// TIA Portal V17 export
// export: Created 2022-02-03T14:45:11.768442Z, ExportSetting WithDefaults, DisplayName Totally Integrated Automation Portal, DisplayVersion V17, DisplayName TIA Portal Openness, DisplayVersion V17, DisplayName TIA Portal Version Control Interface, DisplayVersion V17, DisplayName SINAMICS Startdrive Advanced, DisplayVersion V17, DisplayName SINAMICS Startdrive G130, G150, S120, S150, SINAMICS MV, S210, DisplayVersion V17, DisplayName SINAMICS Startdrive G110M, G120, G120C, G120D, G120P, G115D, DisplayVersion V17, DisplayName STEP 7 Professional, DisplayVersion V17, DisplayName STEP 7 Safety, DisplayVersion V17, DisplayName WinCC Advanced, DisplayVersion V17
FUNCTION_BLOCK "lifeBitControl"   // FB6, LAD
VERSION : 0.1
// stored: Access Published, AutoNumber true, IsIECCheckEnabled false, IsRetainMemResEnabled false, MemoryReserve 100, SetENOAutomatically false, UDAEnableTagReadback false
   VAR_INPUT
      acknowledge : Bool;
   END_VAR
   VAR_OUTPUT
      warning : Bool;
   END_VAR
   VAR
      statTPCoordination : Word;
      IntIEC_Timer1 { S7_SetPoint := 'True'} : TON_TIME;
      InstIEC_Timer2 { S7_SetPoint := 'True'} : TON_TIME;
      statOldAcknowledge { S7_SetPoint := 'True'} : Bool;
      statOldTimer : Bool;
   END_VAR
   VAR_TEMP
      tempTimer1 : Bool;
      tempTimer2 : Bool;
   END_VAR
   VAR_TEMP   // added for the SCL form of the ladder/FBD networks
      _w1 : Bool;
      _w2 : Bool;
      _w3 : Bool;
   END_VAR
BEGIN

REGION Network 1
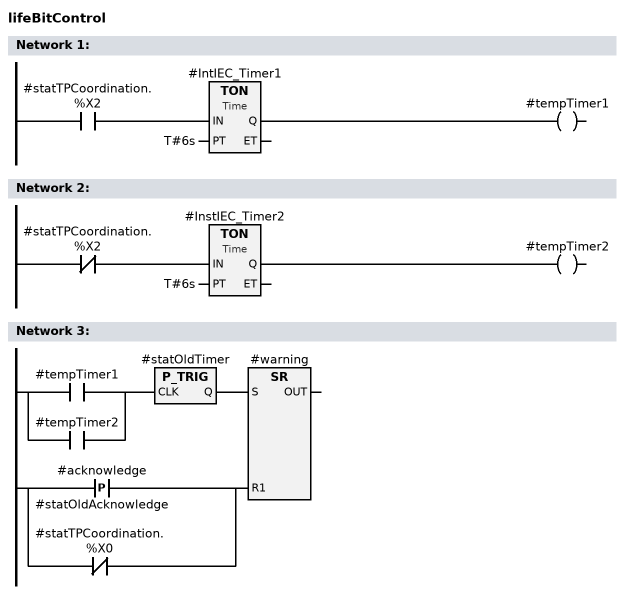
   RUNG wire#powerrail
      Contact( #statTPCoordination.%X2 )
      { S7_Templates := "time_type := Time" } #IntIEC_Timer1.TON(pt := T#6s, et =>)
      Coil( #tempTimer1 )
   END_RUNG
   // the same network as SCL:
   #IntIEC_Timer1(IN := #statTPCoordination.%X2, PT := T#6s);   // TON
   #tempTimer1 := #IntIEC_Timer1.Q;
END_REGION

REGION Network 2
   RUNG wire#powerrail
      I_Contact( #statTPCoordination.%X2 )
      { S7_Templates := "time_type := Time" } #InstIEC_Timer2.TON(pt := T#6s, et =>)
      Coil( #tempTimer2 )
   END_RUNG
   // the same network as SCL:
   #InstIEC_Timer2(IN := NOT #statTPCoordination.%X2, PT := T#6s);   // TON
   #tempTimer2 := #InstIEC_Timer2.Q;
END_REGION

REGION Network 3
   RUNG wire#powerrail
      Contact( #tempTimer1 )
      wire#w1
      P_Trig( #statOldTimer )
      S_SR(operand := #warning, r1 := wire#w2)
   END_RUNG
   RUNG wire#powerrail
      Contact( #tempTimer2 )
   END_RUNG wire#w1
   RUNG wire#powerrail
      P_Contact(operand := #acknowledge, bit := #statOldAcknowledge)
   END_RUNG wire#w2
   RUNG wire#powerrail
      I_Contact( #statTPCoordination.%X0 )
   END_RUNG wire#w2
   // the same network as SCL:
   #_w1 := #tempTimer1 OR #tempTimer2;
   #_w2 := #_w1 AND NOT #statOldTimer;   // rising edge
   #statOldTimer := #_w1;
   #_w3 := #acknowledge AND NOT #statOldAcknowledge;   // rising edge of #acknowledge
   #statOldAcknowledge := #acknowledge;
   IF #_w2 THEN
       #warning := TRUE;   // SR flip-flop
   END_IF;
   IF #_w3 OR NOT #statTPCoordination.%X0 THEN #warning := FALSE; END_IF;
END_REGION
END_FUNCTION_BLOCK
